// Function used in QuickSort
FUNCTION _Partition : DINT
VAR_INPUT
	Arr					: __SYSTEM.AnyType;
	FirstElement		: __SYSTEM.AnyType;
	SortBy				: __SYSTEM.AnyType;
	MemberOffset		: DWORD;
	StartIndex			: DINT; // Starting comparision index
	EndIndex			: DINT; // Ending comparision index
	Order 				: E_Order;
END_VAR
VAR
	Pivot				: POINTER TO BYTE; // Compared number
	Leftwall			: DINT; // New pivot location
	Iterator			: DINT; // For iterator variable
	IterAdr				: POINTER TO BYTE;
	compA				: __SYSTEM.AnyType := SortBy; // get data of compared variable
	compB				: __SYSTEM.AnyType := SortBy;
END_VAR


Pivot := Arr.pValue + FirstElement.diSize * EndIndex;

Leftwall := StartIndex;

FOR Iterator := StartIndex TO EndIndex - 1 DO

	IterAdr := Arr.pValue + FirstElement.diSize * Iterator;
	
	compA.pValue := IterAdr + MemberOffset; // data of compared variable stays the same, just point to other value
	compB.pValue := Pivot + MemberOffset;
	
	CASE Order OF
		E_Order.ASCENDING:
			IF IsLessThanOrEqualAnyType(compA, compB) = E_GeneralResult._TRUE THEN

				SwapByAddr(IterAdr, Arr.pValue + FirstElement.diSize * Leftwall, FirstElement.diSize);
				Leftwall := Leftwall + 1;
			END_IF
		E_Order.DESCENDING:
			IF IsGreaterThanOrEqualAnyType(compA, compB) = E_GeneralResult._TRUE THEN

				SwapByAddr(IterAdr, Arr.pValue + FirstElement.diSize * Leftwall, FirstElement.diSize);
				Leftwall := Leftwall + 1;
			END_IF
	END_CASE
END_FOR

SwapByAddr(Arr.pValue + FirstElement.diSize * Leftwall, Pivot, FirstElement.diSize);

_Partition := Leftwall;

END_FUNCTION

(* stored: Version 1.1.0.1, ProductVersion 3.1.4024.11
   POU _Partition: Id {3ded649f-0755-479b-9bc6-855de8b30060}, SpecialFunc None *)
